// TIA Portal V17 export
// export: Created 2024-06-16T17:47:34.3388825Z, ExportSetting WithDefaults, DisplayName Totally Integrated Automation Portal, DisplayVersion V17, DisplayName TIA Portal Openness, DisplayVersion V17, DisplayName TIA Portal Version Control Interface, DisplayVersion V17, DisplayName STEP 7 Professional, DisplayVersion V17, DisplayName STEP 7 Safety, DisplayVersion V17, DisplayName WinCC Professional, DisplayVersion V17
DATA_BLOCK "St4_Out"   // DB415
{ S7_Optimized_Access := 'TRUE' }
VERSION : 0.1
// stored: AutoNumber false, DBAccessibleFromOPCUA true, DBAccessibleFromWebserver true, IsOnlyStoredInLoadMemory false, IsRetainMemResEnabled false, IsWriteProtectedInAS false, MemoryReserve 100
   VAR
      Sortir_Loquet : Bool;   // Sortir : Loquet (Déplacement Barquette)
      Sortir_PoussoirC : Bool;   // Sortir : Poussoir Z-OK
      Ouverture_PincesC : Bool;   // Ouverture : Pinces C
      Fermeture_PincesC : Bool;   // Fermeture : Pinces C
      Vy_C : Bool;   // Zone Conforme pleine - A vidanger
      Sortir_PoussoirNC : Bool;   // Sortir Poussoir NC
      Ouverture_PincesNC : Bool;   // Ouverture Pinces NC
      Fermeture_PincesNC : Bool;   // Fermeture Pinces NC
      Vy_NC : Bool;   // Zone Non-Conforme pleine - A vidanger
   END_VAR
BEGIN
END_DATA_BLOCK
